{attribute addProperty BoxType "AT2020-0250-0019"}
{attribute addProperty Id "A_0085_AT2050_5500_0018_AT2050_5500AT2050_C5E5984862678.25"}
{attribute addProperty CRC "3735059193"}
{attribute addProperty SizeInBites "626"}
{attribute addProperty SizeInBytes "78.25"}
TYPE A_0060_AT2020_0250_0019_AT2020_0250_DEA07AF9 EXTENDS AT2020_BA5A9548 :
STRUCT
	{attribute addProperty Name "A_0085_AT2050_5500_0018_AT2050_5500"}
	A_0085_AT2050_5500_0018_AT2050_5500 : AT2050_C5E59848;
END_STRUCT
END_TYPE

(* stored: Version 1.2.0.0, ProductVersion 3.1.4024.9
   DUT A_0060_AT2020_0250_0019_AT2020_0250_DEA07AF9: Id {df87f663-53db-4117-9283-6667c5205ac4} *)
